TEXTLIST TL_Nchannel
  0 = 'Choose'
  1 = '2 channels'
  2 = '4 channels'
  3 = '8 channels'
   = ''
END_TEXTLIST

(* stored: Version 1.1.0.1, ProductVersion 3.1.4020.3
   TextList TL_Nchannel: Id {24b2eeb6-941c-4d12-bf37-8045c8f1bfca} *)
